Omron CX-Programmer project 新工程 (CX-Programmer 9.73)

# PLC 新PLC1: CPM2* 

## Program 新程序1 (no task)
; 这个PLC程序实现了一个北人04印刷机的控制系统，应用于印刷厂的印刷生产线。系统通过启动按钮触发工作流程。系统支持通过手动/自动开关进行模式切换。系统包含启动按钮、停止按钮、手动/自动开关、纸张进给传感器、墨水供给传感器、印刷速度传感器。执行器包括印刷机电机控制、纸张进给控制、墨水供给控制、报警灯。 / 操作人员通过手动/自动开关选择运行模式，手动模式由手动模式标志控制，自动模式由自动模式标志控制。但无论何时，手动模式标志和自动模式标志都不会同时为真，以确保操作模式清晰且安全。 / 在自动模式下，按下启动按钮触发流程，但只有在停止按钮未按下时才会开始运行。检测纸张进给状态以监控系统运行情况。系统首先激活纸张进给控制，并通过纸张进给传感器检测状态。如果纸张进给传感器显示异常，系统将点亮报警灯并停止进给，确保纸张进给始终处于正常状态。随后，墨水供给控制启用，并由墨水供给传感器监测状态。 / 序列启动定时器延时30秒控制流程顺序。长时间监测定时器延时300秒进行状态监测。印刷次数计数器1和印刷次数计数器2记录印刷次数，最大值为9999次。状态移位寄存器确保状态按序转移。停止按钮按下时，停止纸张进给控制。若检测到异常，报警灯会亮起，提示操作人员处理故障。
Local symbols
HR BOOL
hr BOOL
il BOOL

### Section 段1

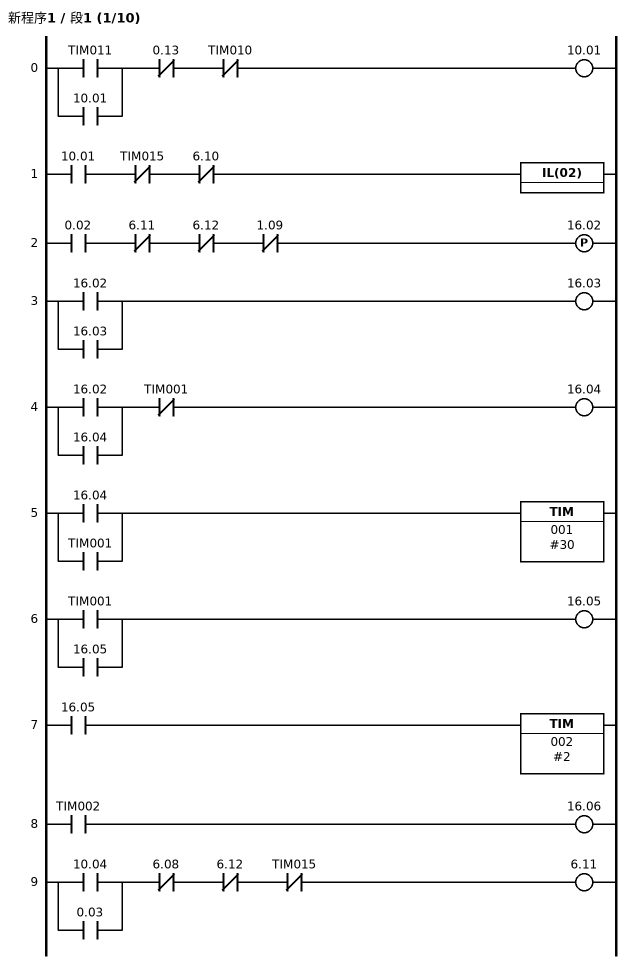
; rung 0
LD TIM011
OR 10.01
ANDNOT 0.13
ANDNOT TIM010
OUT 10.01
; rung 1
LD 10.01
ANDNOT TIM015
ANDNOT 6.10
IL(02)
; rung 2
LD 0.02
ANDNOT 6.11
ANDNOT 6.12
ANDNOT 1.09
DIFU(13) 16.02
; rung 3
LD 16.02
OR 16.03
OUT 16.03
; rung 4
LD 16.02
OR 16.04
ANDNOT TIM001
OUT 16.04
; rung 5
LD 16.04
OR TIM001
TIM 001 #30
; rung 6
LD TIM001
OR 16.05
OUT 16.05
; rung 7
LD 16.05
TIM 002 #2
; rung 8
LD TIM002
OUT 16.06
; rung 9
LD 10.04
OR 0.03
ANDNOT 6.08
ANDNOT 6.12
ANDNOT TIM015
OUT 6.11

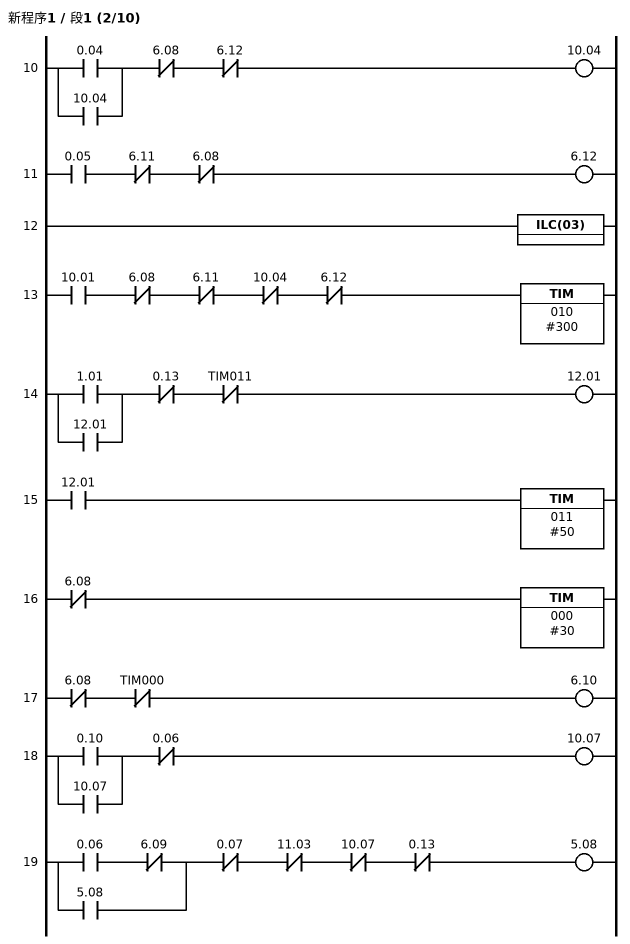
; rung 10
LD 0.04
OR 10.04
ANDNOT 6.08
ANDNOT 6.12
OUT 10.04
; rung 11
LD 0.05
ANDNOT 6.11
ANDNOT 6.08
OUT 6.12
; rung 12
ILC(03)
; rung 13
LD 10.01
ANDNOT 6.08
ANDNOT 6.11
ANDNOT 10.04
ANDNOT 6.12
TIM 010 #300
; rung 14
LD 1.01
OR 12.01
ANDNOT 0.13
ANDNOT TIM011
OUT 12.01
; rung 15
LD 12.01
TIM 011 #50
; rung 16
LDNOT 6.08
TIM 000 #30
; rung 17
LDNOT 6.08
ANDNOT TIM000
OUT 6.10
; rung 18
LD 0.10
OR 10.07
ANDNOT 0.06
OUT 10.07
; rung 19
LD 0.06
ANDNOT 6.09
OR 5.08
ANDNOT 0.07
ANDNOT 11.03
ANDNOT 10.07
ANDNOT 0.13
OUT 5.08

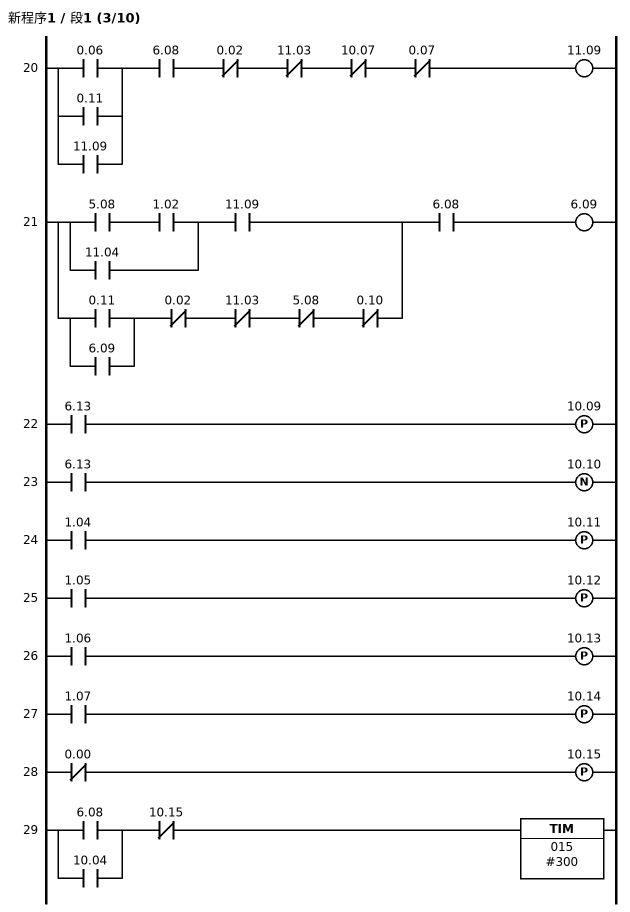
; rung 20
LD 0.06
OR 0.11
OR 11.09
AND 6.08
ANDNOT 0.02
ANDNOT 11.03
ANDNOT 10.07
ANDNOT 0.07
OUT 11.09
; rung 21
LD 5.08
AND 1.02
OR 11.04
AND 11.09
LD 0.11
OR 6.09
ANDNOT 0.02
ANDNOT 11.03
ANDNOT 5.08
ANDNOT 0.10
ORLD
AND 6.08
OUT 6.09
; rung 22
LD 6.13
DIFU(13) 10.09
; rung 23
LD 6.13
DIFD(14) 10.10
; rung 24
LD 1.04
DIFU(13) 10.11
; rung 25
LD 1.05
DIFU(13) 10.12
; rung 26
LD 1.06
DIFU(13) 10.13
; rung 27
LD 1.07
DIFU(13) 10.14
; rung 28
LDNOT 0.00
DIFU(13) 10.15
; rung 29
LD 6.08
OR 10.04
ANDNOT 10.15
TIM 015 #300

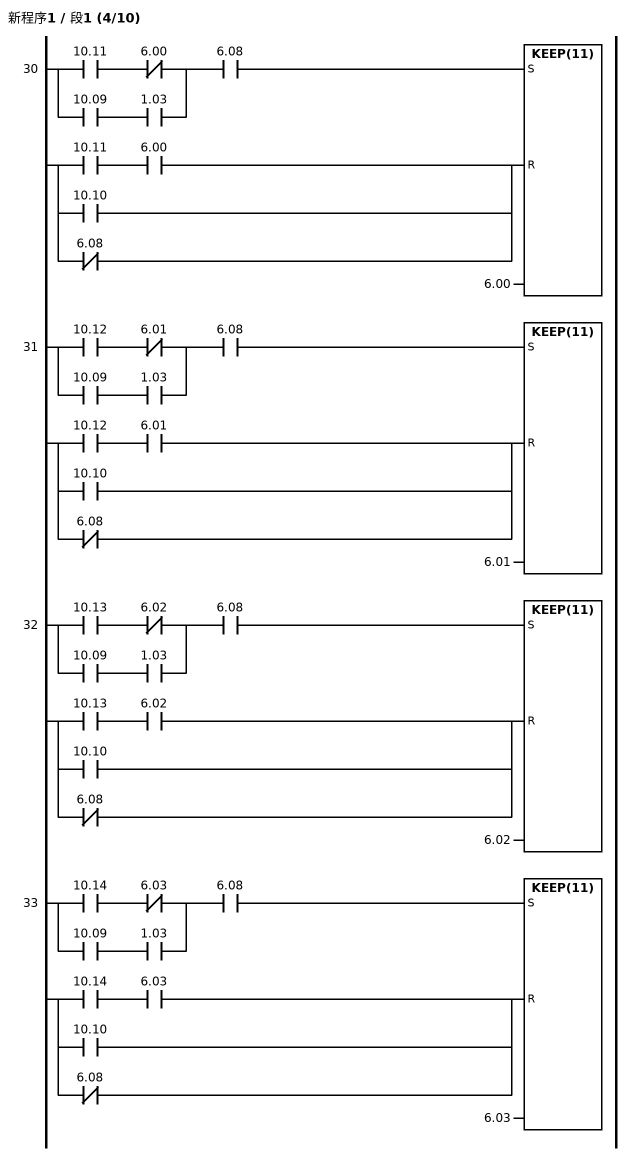
; rung 30
LD 10.11
ANDNOT 6.00
LD 10.09
AND 1.03
ORLD
AND 6.08
LD 10.11
AND 6.00
OR 10.10
ORNOT 6.08
KEEP(11) 6.00
; rung 31
LD 10.12
ANDNOT 6.01
LD 10.09
AND 1.03
ORLD
AND 6.08
LD 10.12
AND 6.01
OR 10.10
ORNOT 6.08
KEEP(11) 6.01
; rung 32
LD 10.13
ANDNOT 6.02
LD 10.09
AND 1.03
ORLD
AND 6.08
LD 10.13
AND 6.02
OR 10.10
ORNOT 6.08
KEEP(11) 6.02
; rung 33
LD 10.14
ANDNOT 6.03
LD 10.09
AND 1.03
ORLD
AND 6.08
LD 10.14
AND 6.03
OR 10.10
ORNOT 6.08
KEEP(11) 6.03

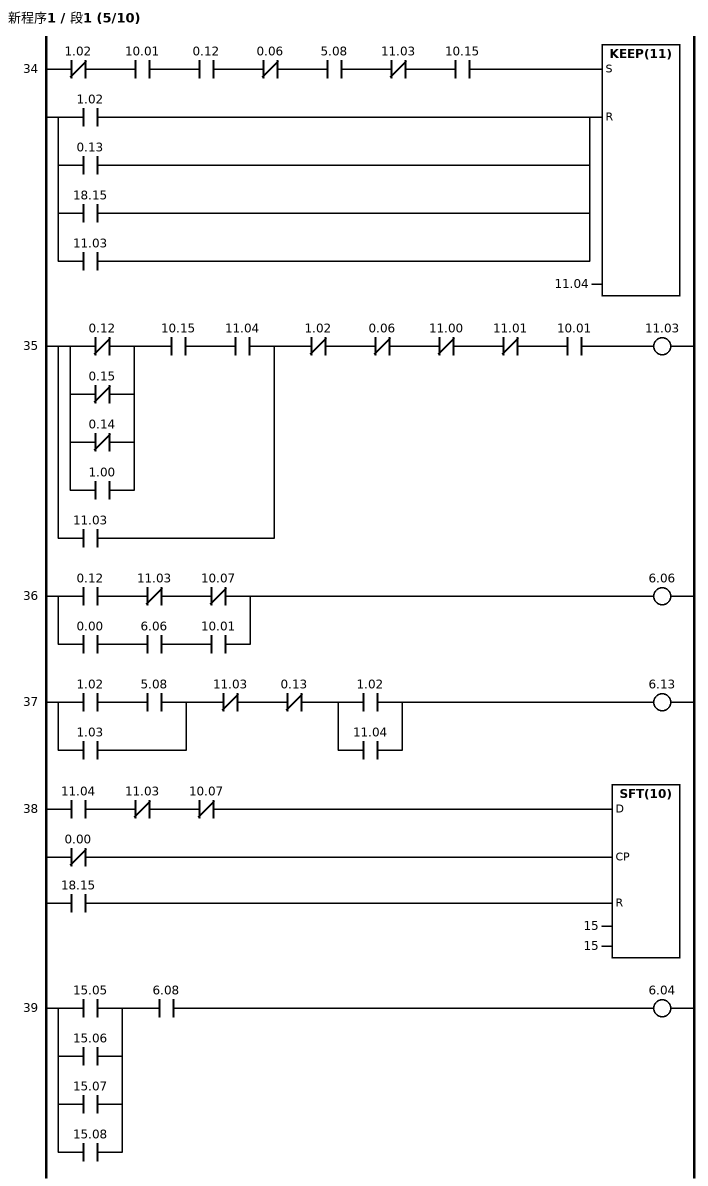
; rung 34
LDNOT 1.02
AND 10.01
AND 0.12
ANDNOT 0.06
AND 5.08
ANDNOT 11.03
AND 10.15
LD 1.02
OR 0.13
OR 18.15
OR 11.03
KEEP(11) 11.04
; rung 35
LDNOT 0.12
ORNOT 0.15
ORNOT 0.14
OR 1.00
AND 10.15
AND 11.04
OR 11.03
ANDNOT 1.02
ANDNOT 0.06
ANDNOT 11.00
ANDNOT 11.01
AND 10.01
OUT 11.03
; rung 36
LD 0.12
ANDNOT 11.03
ANDNOT 10.07
LD 0.00
AND 6.06
AND 10.01
ORLD
OUT 6.06
; rung 37
LD 1.02
AND 5.08
OR 1.03
ANDNOT 11.03
ANDNOT 0.13
LD 1.02
OR 11.04
ANDLD
OUT 6.13
; rung 38
LD 11.04
ANDNOT 11.03
ANDNOT 10.07
LDNOT 0.00
LD 18.15
SFT(10) 15 15
; rung 39
LD 15.05
OR 15.06
OR 15.07
OR 15.08
AND 6.08
OUT 6.04

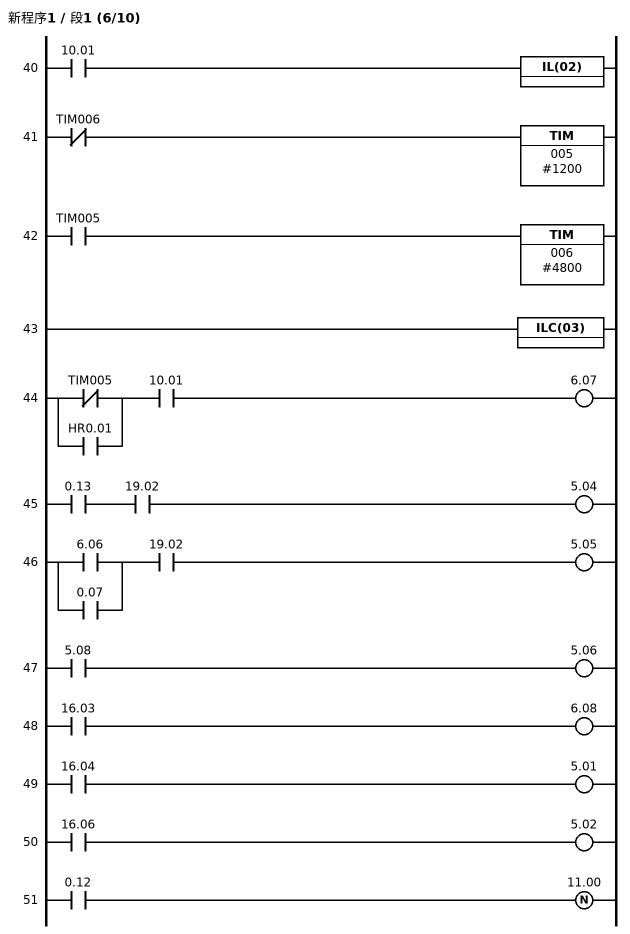
; rung 40
LD 10.01
IL(02)
; rung 41
LDNOT TIM006
TIM 005 #1200
; rung 42
LD TIM005
TIM 006 #4800
; rung 43
ILC(03)
; rung 44
LDNOT TIM005
OR HR0.01
AND 10.01
OUT 6.07
; rung 45
LD 0.13
AND 19.02
OUT 5.04
; rung 46
LD 6.06
OR 0.07
AND 19.02
OUT 5.05
; rung 47
LD 5.08
OUT 5.06
; rung 48
LD 16.03
OUT 6.08
; rung 49
LD 16.04
OUT 5.01
; rung 50
LD 16.06
OUT 5.02
; rung 51
LD 0.12
DIFD(14) 11.00

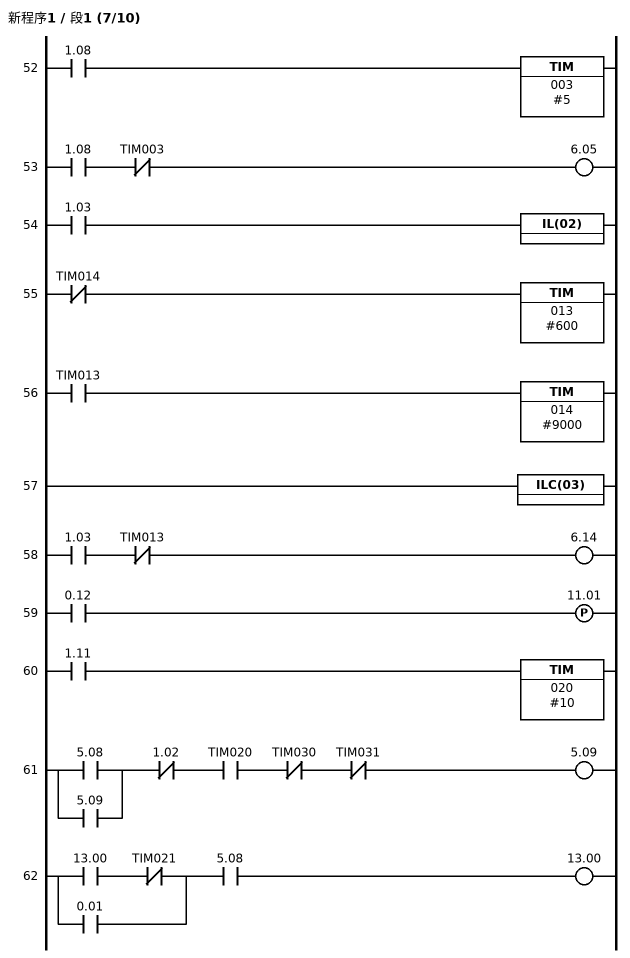
; rung 52
LD 1.08
TIM 003 #5
; rung 53
LD 1.08
ANDNOT TIM003
OUT 6.05
; rung 54
LD 1.03
IL(02)
; rung 55
LDNOT TIM014
TIM 013 #600
; rung 56
LD TIM013
TIM 014 #9000
; rung 57
ILC(03)
; rung 58
LD 1.03
ANDNOT TIM013
OUT 6.14
; rung 59
LD 0.12
DIFU(13) 11.01
; rung 60
LD 1.11
TIM 020 #10
; rung 61
LD 5.08
OR 5.09
ANDNOT 1.02
AND TIM020
ANDNOT TIM030
ANDNOT TIM031
OUT 5.09
; rung 62
LD 13.00
ANDNOT TIM021
OR 0.01
AND 5.08
OUT 13.00

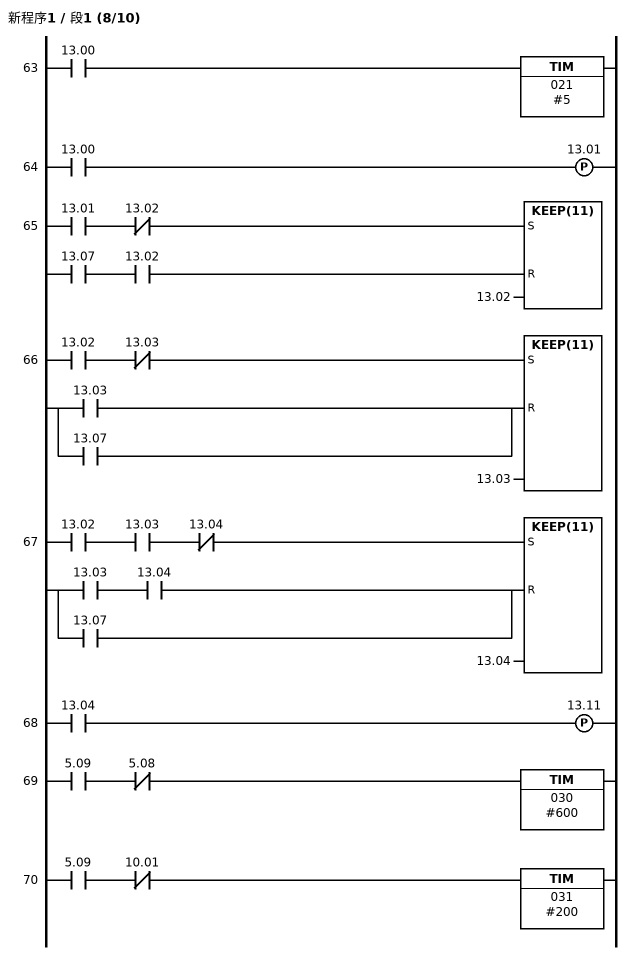
; rung 63
LD 13.00
TIM 021 #5
; rung 64
LD 13.00
DIFU(13) 13.01
; rung 65
LD 13.01
ANDNOT 13.02
LD 13.07
AND 13.02
KEEP(11) 13.02
; rung 66
LD 13.02
ANDNOT 13.03
LD 13.03
OR 13.07
KEEP(11) 13.03
; rung 67
LD 13.02
AND 13.03
ANDNOT 13.04
LD 13.03
AND 13.04
OR 13.07
KEEP(11) 13.04
; rung 68
LD 13.04
DIFU(13) 13.11
; rung 69
LD 5.09
ANDNOT 5.08
TIM 030 #600
; rung 70
LD 5.09
ANDNOT 10.01
TIM 031 #200

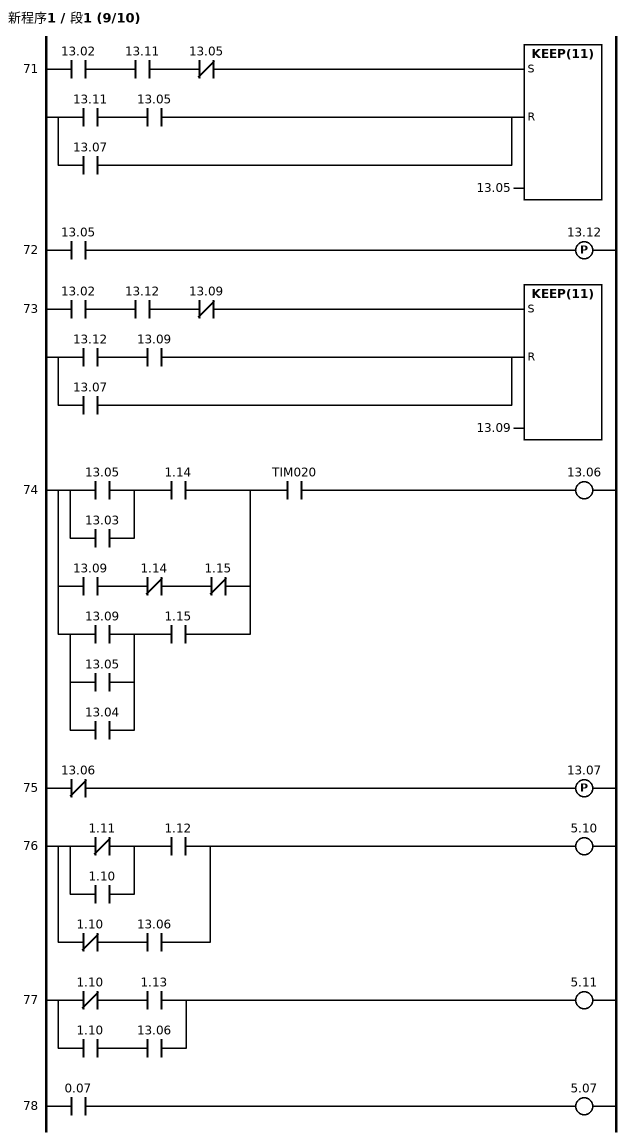
; rung 71
LD 13.02
AND 13.11
ANDNOT 13.05
LD 13.11
AND 13.05
OR 13.07
KEEP(11) 13.05
; rung 72
LD 13.05
DIFU(13) 13.12
; rung 73
LD 13.02
AND 13.12
ANDNOT 13.09
LD 13.12
AND 13.09
OR 13.07
KEEP(11) 13.09
; rung 74
LD 13.05
OR 13.03
AND 1.14
LD 13.09
ANDNOT 1.14
ANDNOT 1.15
ORLD
LD 13.09
OR 13.05
OR 13.04
AND 1.15
ORLD
AND TIM020
OUT 13.06
; rung 75
LDNOT 13.06
DIFU(13) 13.07
; rung 76
LDNOT 1.11
OR 1.10
AND 1.12
LDNOT 1.10
AND 13.06
ORLD
OUT 5.10
; rung 77
LDNOT 1.10
AND 1.13
LD 1.10
AND 13.06
ORLD
OUT 5.11
; rung 78
LD 0.07
OUT 5.07

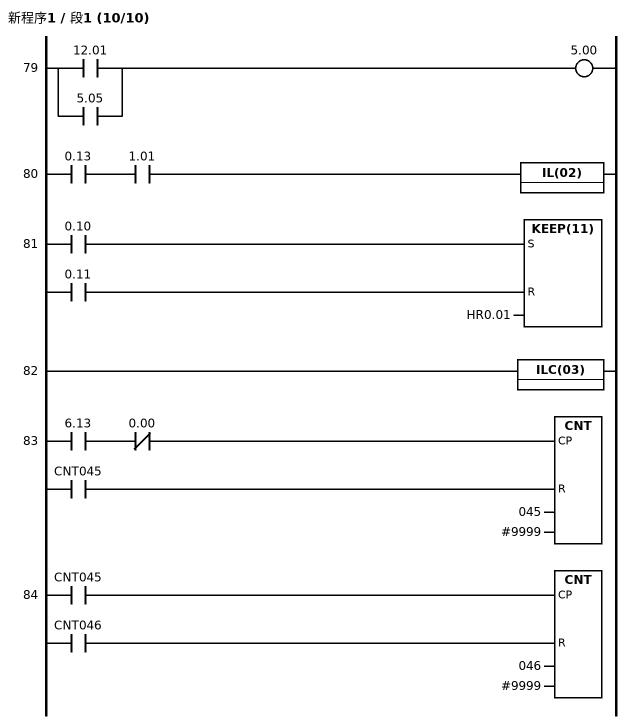
; rung 79
LD 12.01
OR 5.05
OUT 5.00
; rung 80
LD 0.13
AND 1.01
IL(02)
; rung 81
LD 0.10
LD 0.11
KEEP(11) HR0.01
; rung 82
ILC(03)
; rung 83
LD 6.13
ANDNOT 0.00
LD CNT045
CNT 045 #9999
; rung 84
LD CNT045
LD CNT046
CNT 046 #9999
; rung 85
END(01)

### Section 段2
; rung 0
END(01)